(* IEC 61131-3 sources: com.logicals.lc3.webinar/usRTS_RPMControl_iSOC/src_FB_LIB_SAFE/Compare/DWORD, 2 files *)

(* ---- wEQ_DWORD_2.iecst ---- *)
NAMESPACE logicals.web.standard
NAMESPACE compare

/*
 * Function block wrapper for IEC 61131-3 EQ<br>
 * IN1 =  1st value (DWORD)<br>
 * IN2 =  2nd value (DWORD)<br>
 * OUT = true if IN1 is equal to IN2 (BOOL)<br>
 */
FUNCTION_BLOCK wEQ_DWORD_2
	{ vNameAlignment:="center"; altName:="="; bgColor:="DodgerBlue"; width:=40; hideIONames; }
	VAR_INPUT
		IN1 : DWORD;
		IN2 : DWORD;
	END_VAR
	VAR_OUTPUT
		OUT : BOOL;
	END_VAR

	OUT := EQ(IN1:=IN1, IN2:=IN2, ENO=>ENO);
END_FUNCTION_BLOCK

END_NAMESPACE
END_NAMESPACE

(* ---- wNE_DWORD.iecst ---- *)
NAMESPACE logicals.web.standard
NAMESPACE compare

/*
 * Function block wrapper for IEC 61131-3 NE<br>
 * IN1 = value 1 (DWORD)<br>
 * IN2 = value 2 (DWORD)<br>
 * OUT = true if IN1 is not equal to IN2 (BOOL)<br>
 */
FUNCTION_BLOCK wNE_DWORD
	{ vNameAlignment:="center"; altName:="<>"; bgColor:="DodgerBlue"; width:=40; hideIONames; }
	VAR_INPUT
		IN1 : DWORD;
		IN2 : DWORD;
	END_VAR
	VAR_OUTPUT
		OUT : BOOL;
	END_VAR

	OUT := NE(IN1:=IN1, IN2:=IN2, ENO=>ENO);
END_FUNCTION_BLOCK

END_NAMESPACE
END_NAMESPACE
